//Function block to run a virtual drive with Nc
FUNCTION_BLOCK FB_Axis IMPLEMENTS I_axis
VAR
    _stAxis: REFERENCE TO ST_AxisStruct; // Local property pointer for axis structure
    astMcStatus: ARRAY[1..nMCSTATUS_ARRAY_SIZE] OF POINTER TO ST_McStatus; //Array of all MC status signals defined in FB_init

    fbPower: MC_Power;
    stMcStatusPower: ST_McStatus;

    fbStop: MC_Stop;
    stMcStatusStop: ST_McStatus;

    fbHalt: MC_Halt;
    stMcStatusHalt: ST_McStatus;

    fbReset: MC_Reset;
    stMcStatusReset: ST_McStatus;

    //SERCOS drive
    fbSoEReadDiagNumber : FB_SoEReadDiagNumber;
    fbSoEReset: FB_SoEReset;

    fbReadDriveInfo: FB_ReadDriveInfo;

    fbMoveAbsolute: MC_MoveAbsolute;
    fbMoveAbsolute2: MC_MoveAbsolute;
    stMcStatusMoveAbsolute: ST_McStatus;

    fbMoveRelative: MC_MoveRelative;
    stMcStatusMoveRelative: ST_McStatus;

    fbMoveVelocity: MC_MoveVelocity;
    stMcStatusMoveVelocity: ST_McStatus;

    fbMoveModulo: MC_MoveModulo;
    fbMoveModulo2: MC_MoveModulo;
    stMcStatusMoveModulo: ST_McStatus;

    fbBacklashCompensation: MC_BacklashCompensation;
    stMcStatusBacklash: ST_McStatus;

    fbHome: FB_Homing;
    stMcStatusHome: ST_McStatus;

    fbReadParameter: MC_ReadParameter;
    stMcStatusReadParameter: ST_McStatus;

    fbWriteParameter: MC_WriteParameter;
    stMcStatusWriteParameter: ST_McStatus;

    stMcStatusReadWriteCoE: ST_McStatus;
    fb_coe_writeEx: FB_EcCoESdoWriteEx; // Function Block for writing in CoE
    fb_coe_readEx: FB_EcCoESdoReadEx;  // Function Block for reading from CoE

    fbGearIn: MC_GearIn;
    stMcStatusGearIn: ST_McStatus;

    fbGearOut: MC_GearOut;
    stMcStatusGearOut: ST_McStatus;

    stMasterAxis: ST_GearAxis := (nIndex := 1, fRatio := 0);
    nSlaveAxesIndex: UINT;
    nAxisIndex: UINT;
    nMultiMastersAxesIndex: UINT;

    fbGearInMultiMaster: MC_GearInMultiMaster;
    stMcStatusGearInMultiMaster: ST_McStatus;

    //Custom made methods MC Status
    stMcStatusTempDisable: ST_McStatus;
    stMcStatusCommandHandler: ST_McStatus;
    stMcStatusAirpad: ST_McStatus;
    stMcStatusExternalBrake: ST_McStatus;

    //Variables for holding limits during homing
    bWaitForStopAfterLimitHit: BOOL := FALSE;
    fbRemovePowerTimer: TOF;

    //Dedicated NC parameter read FBs
    fbReadAxisVeloManSlow: MC_ReadParameter;
    fbReadAxisVeloManFast: MC_ReadParameter;
    fbReadHomingVelToCam: MC_ReadParameter;
    fbReadHomingVelFromCam: MC_ReadParameter;
    fbReadAxisVeloMax: MC_ReadParameter;
    fbReadAxisMaxAcc: MC_ReadParameter;
    fbReadAxisMaxDec: MC_ReadParameter;
    fbReadAxisAcc: MC_ReadParameter;
    fbReadAxisDec: MC_ReadParameter;
    fbReadEnMinSoftPosLimit: MC_ReadParameter;
    fbReadEnMaxSoftPosLimit: MC_ReadParameter;
    fbReadMinSoftPosLimit: MC_ReadParameter;
    fbReadMaxSoftPosLimit: MC_ReadParameter;
    fbReadEnPositionLagMonitoring: MC_ReadParameter;
    fbReadAxisMaxPosLagValue: MC_ReadParameter;
    fbReadEnTargetPositionMonitoring: MC_ReadParameter;
    fbReadTargetPositionWindow: MC_ReadParameter;
    fbReadBacklashConfigEnable: MC_ReadParameter;
    fbReadDriveAdress: MC_ReadDriveAddress;

    //Edge detection triggers for statuses
    fbDoneRTrig: R_TRIG;
    fbCommandAbortedRTrig: R_TRIG;
    fbInVelocityRTrig: R_TRIG;
    fbInVelocityFTrig: F_TRIG;
    fbExecuteRTrig: R_TRIG;
    fbStopFinishedRiseEdge: R_TRIG;
    fbHaltFinishedRiseEdge: R_TRIG;
    fbResetFinishedRiseEdge: R_TRIG;
    fbAbsMovDyn1RiseEdge: R_TRIG;
    fbAbsMovDyn2RiseEdge: R_TRIG;
    fbModMovDyn1RiseEdge: R_TRIG;
    fbModMovDyn2RiseEdge: R_TRIG;

    fbCommandHistory: FB_CommandHistory;

    bInternalExecute: BOOL := FALSE;
    bEnableCmdOld: BOOL := FALSE;
    bEnabledOld: BOOL := FALSE;
    bEnableAmpCmd: BOOL := FALSE;
END_VAR

VAR CONSTANT
    nRATIO_DENOMINATOR_DEFAULT: UINT := 1;
    nNO_GEARING: UINT := 0;
    nFIRST_ARRAY_INDEX_MOVE_COMMANDS: UINT := 5; //Used for the FOR loops for the Busy, Done, Command Aborted Status
    nLAST_ARRAY_INDEX_MOVE_COMMANDS: UINT := 15; //Used for the FOR loops for Done
    nMCSTATUS_ARRAY_SIZE: UINT := 19;
    nMULTI_MASTER_MAX_AXES: UINT := 4;
END_VAR

METHOD EndOfCycle : BOOL
IF _stAxis.stStatus.bDone
    OR _stAxis.stStatus.bError
    OR _stAxis.Axis.Status.Error
    OR _stAxis.Axis.Status.Disabled
    OR _stAxis.Axis.Status.Stopping
    OR _stAxis.stStatus.bCommandAborted
    OR NOT _stAxis.stStatus.bMoving THEN
    _stAxis.stStatus.eInternalMotionCommand := E_MotionFunctions.eWaitingForCommand;
END_IF

bInternalExecute := FALSE;
bEnabledOld := _stAxis.stStatus.bEnabled;
bEnableCmdOld := _stAxis.stControl.bEnable;

_stAxis.stControl.bExecute := FALSE;
END_METHOD

METHOD FB_init : BOOL
VAR_INPUT
    bInitRetains: BOOL; // if TRUE, the retain variables are initialized (warm start / cold start)
    bInCopyCode: BOOL; // if TRUE, the instance afterwards gets moved into the copy code (online change)
END_VAR
//Copy address locations for statuses to an array to allow for easier checking of statuses
astMcStatus[1] := ADR(stMcStatusPower);
astMcStatus[2] := ADR(stMcStatusStop);
astMcStatus[3] := ADR(stMcStatusHalt);
astMcStatus[4] := ADR(stMcStatusReset);
astMcStatus[5] := ADR(stMcStatusMoveAbsolute);
astMcStatus[6] := ADR(stMcStatusMoveRelative);
astMcStatus[7] := ADR(stMcStatusMoveVelocity);
astMcStatus[8] := ADR(stMcStatusMoveModulo);
astMcStatus[9] := ADR(stMcStatusHome);
astMcStatus[10] := ADR(stMcStatusGearInMultiMaster);
astMcStatus[11] := ADR(stMcStatusGearOut);
astMcStatus[12] := ADR(stMcStatusReadParameter);
astMcStatus[13] := ADR(stMcStatusWriteParameter);
astMcStatus[14] := ADR(stMcStatusReadWriteCoE);
astMcStatus[15] := ADR(stMcStatusBacklash);
astMcStatus[16] := ADR(stMcStatusTempDisable);
astMcStatus[17] := ADR(stMcStatusCommandHandler);
astMcStatus[18] := ADR(stMcStatusAirpad);
astMcStatus[19] := ADR(stMcStatusExternalBrake);
END_METHOD

// Controls pressure to airpad
METHOD mControl_Airpad : ST_McStatus
VAR_INPUT
    bMoveRequest: BOOL;
    bManualControl: BOOL;
    bManualPressureOn: BOOL;
END_VAR

VAR_OUTPUT
    bReady: BOOL;
END_VAR

VAR_INST
    eAirpad: E_Airpad := E_Airpad.eDepressurize;
    TON_PressurizeAirpad: TON;
    TON_Depressurize: TON;
    RTRIG_PressureRequest: R_TRIG;
    bNotPressurizedInTime: BOOL := FALSE;
    bPressureOnRequest: BOOL := FALSE;
    RTRIG_ManualControl: R_TRIG;

    nAirpadErrorId: UDINT := 0;
END_VAR
IF NOT _stAxis.stConfig.stAirpadBrake.bAirpadConnected THEN
    RETURN;
END_IF

RTRIG_ManualControl(CLK := _stAxis.stConfig.bAirpadManualControl);

IF RTRIG_ManualControl.Q THEN
    _stAxis.stControl.bAirpadManualPressureOn := bMoveRequest;
ELSIF NOT _stAxis.stConfig.bAirpadManualControl THEN
    _stAxis.stControl.bAirpadManualPressureOn := FALSE;
END_IF

bPressureOnRequest :=
    (bMoveRequest
        AND NOT bManualControl)
    OR (bManualControl
        AND bManualPressureOn);

RTRIG_PressureRequest(CLK := bPressureOnRequest);

TON_PressurizeAirpad(
    IN := bPressureOnRequest
        AND NOT _stAxis.stStatus.bError,
    PT := _stAxis.stConfig.stAirpadBrake.tAirpadOnDelayTime);

TON_Depressurize(
    IN := NOT bPressureOnRequest,
    PT := _stAxis.stConfig.stAirpadBrake.tAirpadOffDelayTime);

CASE eAirpad OF

    E_Airpad.eDepressurize:
        //No movement requested -> Airpad off
        _stAxis.stControl.bPressurizeAirpad := FALSE;
        IF bPressureOnRequest
            AND NOT _stAxis.stStatus.bError
            AND NOT _stAxis.stStatus.bAirpadPressureError THEN
            _stAxis.stStatus.bAirpadPressureError := FALSE;
            nAirpadErrorId := 0;
            eAirpad := E_Airpad.ePressurize;
        END_IF


    E_Airpad.ePressurize:
        //Movement requested -> Pressurize airpad
        _stAxis.stControl.bPressurizeAirpad := TRUE;

        IF _stAxis.stStatus.bError
            OR NOT bPressureOnRequest
            OR _stAxis.stStatus.bAirpadPressureError THEN
            eAirpad := E_Airpad.eDepressurize;
        ELSIF TON_PressurizeAirpad.Q THEN
            IF _stAxis.stConfig.stAirpadBrake.bAirpadFeedbackConnected
                AND NOT _stAxis.stInputs.bAirpadPressurized THEN
                _stAxis.stStatus.bAirpadPressureError := TRUE;
                nAirpadErrorId := E_CustomErrorIds.eAirPadPressureError;
                eAirpad := E_Airpad.eDepressurize;
            ELSE
                eAirpad := E_Airpad.eReadyToMove;
            END_IF
        END_IF


    E_Airpad.eReadyToMove:
        //Movement requested -> Airpad inflated
        _stAxis.stControl.bPressurizeAirpad := TRUE;

        IF _stAxis.stStatus.bError
            OR TON_Depressurize.Q
            OR _stAxis.stStatus.bAirpadPressureError THEN
            eAirpad := E_Airpad.eDepressurize;
        ELSIF (_stAxis.stConfig.stAirpadBrake.bAirpadFeedbackConnected
            AND NOT _stAxis.stInputs.bAirpadPressurized) THEN
            _stAxis.stStatus.bAirpadPressureError := TRUE;
            nAirpadErrorId := E_CustomErrorIds.eAirPadPressureError;
            eAirpad := E_Airpad.eDepressurize;
        END_IF

END_CASE

bReady := eAirpad = E_Airpad.eReadyToMove
    AND ((_stAxis.stConfig.stAirpadBrake.bAirpadFeedbackConnected
        AND _stAxis.stInputs.bAirpadPressurized)
    OR NOT _stAxis.stConfig.stAirpadBrake.bAirpadFeedbackConnected);

//ST_McStatus mapping
mControl_Airpad.Error := _stAxis.stStatus.bAirpadPressureError;
mControl_Airpad.ErrorID := nAirpadErrorId;

IF _stAxis.stStatus.bAirpadPressureError THEN
    _stAxis.stError.nAirpadErrorID := nAirpadErrorId;
END_IF
END_METHOD

METHOD mControl_BacklashCompensation : ST_McStatus
VAR_INPUT
END_VAR
(*Read Backlash documentation in the Confluence page or in Beckhoff before backlash setup:
https://confluence.ess.eu/display/MCAG/Backlash+compensation
Position compensation needs to be enabled in NC to use the backsash compensation*)

IF _stAxis.stConfig.stBacklashConfig.bEnabledInNC THEN

// Enabling the backlash functionality. It is disable if homing is performed.
    IF _stAxis.stStatus.bEnabled THEN
        IF fbHome.bBusy THEN
            fbBacklashCompensation.Enable := FALSE;
        ELSE
            fbBacklashCompensation.Enable := _stAxis.stConfig.stBacklashConfig.bEnableCompensation;
        END_IF
        fbBacklashCompensation.Backlash := _stAxis.stConfig.stBacklashConfig.fCorrectionSetting;
        fbBacklashCompensation.CompensationInPositiveDirection := _stAxis.stConfig.stBacklashConfig.bCompensationInPositiveDirection;
        fbBacklashCompensation.Ramp := ABS(_stAxis.stControl.fVelocity/3);
    ELSE
        fbBacklashCompensation.Enable := FALSE;
        fbBacklashCompensation.DisableMode := 1;
    END_IF

    fbBacklashCompensation(Axis := _stAxis.Axis);

END_IF

IF fbBacklashCompensation.Error THEN
    _stAxis.stError.nBacklashErrorID := fbBacklashCompensation.ErrorID;
END_IF
mControl_BacklashCompensation.Error := fbBacklashCompensation.Error;
mControl_BacklashCompensation.ErrorID := fbBacklashCompensation.ErrorID;
_stAxis.stStatus.bBacklashCompensating := fbBacklashCompensation.Limiting;
END_METHOD

// Handles delayed execution of motion commands due to e.g. auto-enable, airpad or external brake
METHOD mControl_CommandHandler : ST_McStatus

VAR_INPUT
    bAxisPermittedToMove: BOOL := FALSE;
    bPermitRequired: BOOL := FALSE;
END_VAR

VAR_OUTPUT
    bWaitingForMovePermit: BOOL;
    bMovePermit: BOOL;
    bReleaseMoveCmd: BOOL;
END_VAR

VAR
    bCommandAborted: BOOL;
END_VAR

VAR_INST
    eState: E_CommandHandlerState := E_CommandHandlerState.eIdle;
    eLatchedCommand: E_MotionFunctions;
    bInternalWaitingForMovePermit: BOOL := FALSE;
    bInternalMovePermit: BOOL := FALSE;
    bInternalReleasedMoveCmd: BOOL := FALSE;
    nWaitCounter: UINT := 0;
    RTRIG_Execute: R_TRIG;
    FTRIG_Moving: F_TRIG;
    TON_CommandHandlerTimeout: TON;
    RTRIG_ReleasedMoveCommand: R_TRIG;
    TON_LatchReleasedCommandStatus: TON;
    TON_DisableAxis: TON;
    RTRIG_DisableAxis: R_TRIG;
END_VAR
//State machine for command handling
RTRIG_Execute(CLK := _stAxis.stControl.bExecute);
RTRIG_ReleasedMoveCommand(CLK := bInternalReleasedMoveCmd);

CASE eState OF
    E_CommandHandlerState.eIdle:
        IF RTRIG_Execute.Q THEN
            CASE _stAxis.stControl.eCommand OF
                E_MotionFunctions.eMoveAbsolute,
                E_MotionFunctions.eMoveRelative,
                E_MotionFunctions.eMoveVelocity,
                E_MotionFunctions.eMoveModulo,
                E_MotionFunctions.eGearInMultiMaster,
                E_MotionFunctions.eGearOut,
                E_MotionFunctions.eHome :
                    eLatchedCommand := _stAxis.stControl.eCommand;
                    nWaitCounter := 0;
                    _stAxis.stStatus.bCommandHandlerTimeoutError := FALSE;

                    IF _stAxis.stConfig.bAutoEnable THEN
                        _stAxis.stControl.bEnable := TRUE;
                    END_IF

                    fbCommandHistory.mAdd(_stAxis.stControl);
                    eState := E_CommandHandlerState.eWaitPermits;
            END_CASE
        END_IF

    E_CommandHandlerState.eWaitPermits:
        IF (bPermitRequired AND bAxisPermittedToMove)
            OR NOT bPermitRequired
            OR (bPermitRequired AND NOT _stAxis.stConfig.bAutoEnable AND NOT _stAxis.stStatus.bEnabled) THEN

            eState := E_CommandHandlerState.eStabilizeNC;
        END_IF

    E_CommandHandlerState.eStabilizeNC:
        //Ensure permits are still valid during stabilization
        IF (bPermitRequired AND NOT bAxisPermittedToMove) THEN
             eState := E_CommandHandlerState.eWaitPermits;
             nWaitCounter := 0;
        ELSIF nWaitCounter >= _stAxis.stConfig.nCommandHandlerWaitCycles THEN
            eState := E_CommandHandlerState.eReleaseCommand;
        ELSE
            nWaitCounter := nWaitCounter + 1;
        END_IF

    E_CommandHandlerState.eReleaseCommand:
        _stAxis.stStatus.eInternalMotionCommand := eLatchedCommand;
        bInternalExecute := TRUE;
        bInternalMovePermit := TRUE;
        bInternalReleasedMoveCmd := TRUE;
        fbCommandHistory.mSetRelease();
        eState := E_CommandHandlerState.eWaitForMotionStart;

    E_CommandHandlerState.eWaitForMotionStart:
        IF _stAxis.stStatus.bMoving
            OR _stAxis.stStatus.bDone
            OR _stAxis.stStatus.bError THEN
            eState := E_CommandHandlerState.eIdle;
        END_IF

END_CASE

bInternalWaitingForMovePermit := (eState = E_CommandHandlerState.eWaitPermits OR eState = E_CommandHandlerState.eStabilizeNC);

TON_CommandHandlerTimeout(
    IN := bInternalWaitingForMovePermit,
    PT := _stAxis.stConfig.tCommandHandlerTimeout);

TON_LatchReleasedCommandStatus(IN := bInternalReleasedMoveCmd, PT := T#1S);

IF TON_CommandHandlerTimeout.Q THEN
    eState := E_CommandHandlerState.eIdle;
    bInternalWaitingForMovePermit := FALSE;
    bInternalMovePermit := FALSE;
    bInternalReleasedMoveCmd := FALSE;
    _stAxis.stStatus.bCommandHandlerTimeoutError := TRUE;
END_IF

IF _stAxis.stControl.bHalt
    OR _stAxis.stControl.bStop THEN
    bCommandAborted := bInternalWaitingForMovePermit;
    eState := E_CommandHandlerState.eIdle;
    bInternalWaitingForMovePermit := FALSE;
    bInternalMovePermit := FALSE;
    bInternalReleasedMoveCmd := FALSE;
END_IF

FTRIG_Moving(CLK :=
    (_stAxis.stStatus.bMoving AND NOT _stAxis.Axis.Status.HomingBusy)
    OR _stAxis.Axis.Status.HomingBusy);

IF FTRIG_Moving.Q
    OR _stAxis.stStatus.bError THEN
    eState := E_CommandHandlerState.eIdle;
    bInternalWaitingForMovePermit := FALSE;
    bInternalMovePermit := FALSE;
    bInternalReleasedMoveCmd := FALSE;
END_IF

TON_DisableAxis(
    IN := _stAxis.stConfig.bAutoDisable
        AND _stAxis.stStatus.bEnabled
        AND NOT bInternalWaitingForMovePermit
        AND NOT bInternalMovePermit
        AND NOT bInternalReleasedMoveCmd,
    PT := _stAxis.stConfig.tAutoDisableHysteresis);
RTRIG_DisableAxis(CLK := TON_DisableAxis.Q);
IF RTRIG_DisableAxis.Q
    AND _stAxis.stConfig.bAutoDisable THEN
    _stAxis.stControl.bEnable := FALSE;
END_IF

IF RTRIG_ReleasedMoveCommand.Q THEN
    bInternalReleasedMoveCmd := TRUE;
END_IF

IF TON_LatchReleasedCommandStatus.Q THEN
    bInternalReleasedMoveCmd := FALSE;
END_IF

bWaitingForMovePermit := bInternalWaitingForMovePermit;
bMovePermit := bInternalMovePermit;
bReleaseMoveCmd := bInternalReleasedMoveCmd;

mControl_CommandHandler.CommandAborted := bCommandAborted;
mControl_CommandHandler.Done := bInternalExecute;
mControl_CommandHandler.Busy := (eState <> E_CommandHandlerState.eIdle);
mControl_CommandHandler.Error := _stAxis.stStatus.bCommandHandlerTimeoutError;

IF _stAxis.stStatus.bCommandHandlerTimeoutError THEN
    mControl_CommandHandler.ErrorID := TO_UDINT(E_CustomErrorIds.eCommandHandlerTimeoutError);
    _stAxis.stError.nCommandHandlerErrorID := mControl_CommandHandler.ErrorID;
END_IF
END_METHOD

// Controls external brake
METHOD mControl_ExternalBrake: BOOL

VAR_OUTPUT
    bReady: BOOL;
END_VAR

VAR_INST
    eExternalBrake: E_ExternalBrake := E_ExternalBrake.eBrakeEngaged;
    bEnableAmp: BOOL := FALSE;
    TON_DelayBrakeRelease: TON;
    TON_DelayAmplifierDisable: TON;
    bStartDelayBrakeOpening: BOOL := FALSE;
    bStartDelayAmplifierDisable: BOOL := FALSE;
    bStartBrakeOpeningTimeout: BOOL := FALSE;
    TON_BrakeOpeningTimeoutWhenFeedback: TON;
END_VAR
IF _stAxis.stControl.bEnable AND NOT bEnableCmdOld
    AND NOT _stAxis.stStatus.bExternalBrakeFailure THEN
    eExternalBrake := E_ExternalBrake.eDelayBrakeRelease;
    bStartDelayBrakeOpening := FALSE;
    _stAxis.stStatus.bExternalBrakeTimeoutError  := FALSE;
END_IF

IF (NOT _stAxis.stControl.bEnable OR _stAxis.stStatus.bError)
    AND bEnableCmdOld THEN
    eExternalBrake := E_ExternalBrake.eCloseBrakeDelayAmplifier;
    bStartDelayAmplifierDisable := FALSE;
END_IF

TON_DelayBrakeRelease(
    IN := bStartDelayBrakeOpening,
    PT := _stAxis.stConfig.stAirpadBrake.tBrakeOpenDelayTime
);

TON_DelayAmplifierDisable(
    IN := bStartDelayAmplifierDisable,
    PT := _stAxis.stConfig.stAirpadBrake.tBrakeCloseAheadTime
);

TON_BrakeOpeningTimeoutWhenFeedback(
    IN := bStartBrakeOpeningTimeout,
    PT := _stAxis.stConfig.stAirpadBrake.tBrakeOpeningTimeoutWhenFeedback
);

IF TON_BrakeOpeningTimeoutWhenFeedback.Q THEN
    _stAxis.stStatus.bExternalBrakeTimeoutError := TRUE;
END_IF

CASE eExternalBrake OF

    E_ExternalBrake.eBrakeEngaged:
        _stAxis.stControl.bReleaseBrake := FALSE;
        bStartDelayBrakeOpening := FALSE;
        bStartDelayAmplifierDisable := FALSE;
        bStartBrakeOpeningTimeout := FALSE;
        bEnableAmp := FALSE;


    E_ExternalBrake.eDelayBrakeRelease:
        // Postpone opening of brake
        bEnableAmp := TRUE;
        bStartDelayAmplifierDisable := FALSE;

        IF TON_DelayBrakeRelease.Q THEN
            IF NOT _stAxis.stStatus.bEnabled
                OR _stAxis.stStatus.bError
                OR TON_BrakeOpeningTimeoutWhenFeedback.Q THEN
                _stAxis.stControl.bEnable := FALSE;
                _stAxis.stControl.bReleaseBrake := FALSE;
                bEnableAmp := FALSE;
                eExternalBrake := E_ExternalBrake.eBrakeEngaged;
            ELSE
                _stAxis.stControl.bReleaseBrake := TRUE;
                bStartBrakeOpeningTimeout := TRUE;
            END_IF

            IF _stAxis.stControl.bReleaseBrake
                AND ((_stAxis.stConfig.stAirpadBrake.bExternalBrakeFeedbackConnected
                    AND _stAxis.stInputs.bBrakeReleased)
                OR NOT _stAxis.stConfig.stAirpadBrake.bExternalBrakeFeedbackConnected) THEN
                eExternalBrake := E_ExternalBrake.eBrakeReleased;
                bStartBrakeOpeningTimeout := FALSE;
            END_IF
        END_IF

        // If enabled lost while opening, go directly to closed
        IF bEnabledOld
            AND (NOT _stAxis.stStatus.bEnabled OR _stAxis.stStatus.bError) THEN
            eExternalBrake := E_ExternalBrake.eBrakeEngaged;
            bEnableAmp := FALSE;
            _stAxis.stControl.bReleaseBrake := FALSE;
        END_IF

        // Start counting when enabled
        IF _stAxis.stStatus.bEnabled
            AND eExternalBrake <> E_ExternalBrake.eBrakeReleased THEN
            bStartDelayBrakeOpening := TRUE;
        END_IF


    E_ExternalBrake.eBrakeReleased:
        bStartDelayBrakeOpening := FALSE;
        bStartDelayAmplifierDisable := FALSE;
        // If enabled lost, or if brake feedback fails: go directly to closed
        IF (NOT _stAxis.stStatus.bEnabled OR _stAxis.stStatus.bError)
            AND _stAxis.stControl.bEnable THEN
            _stAxis.stControl.bReleaseBrake := FALSE;
            _stAxis.stControl.bEnable := FALSE;
            bEnableAmp := FALSE;
            eExternalBrake := E_ExternalBrake.eBrakeEngaged;
        ELSIF _stAxis.stConfig.stAirpadBrake.bExternalBrakeFeedbackConnected
            AND _stAxis.stControl.bReleaseBrake
            AND NOT _stAxis.stInputs.bBrakeReleased THEN
            _stAxis.stControl.bReleaseBrake := FALSE;
            _stAxis.stControl.bEnable := FALSE;
            bEnableAmp := FALSE;
            eExternalBrake := E_ExternalBrake.eBrakeEngaged;
            _stAxis.stStatus.bExternalBrakeFailure := TRUE;
        ELSE
            _stAxis.stControl.bReleaseBrake := TRUE;
            bEnableAmp := TRUE;
        END_IF


    // The check for bError in first rows of this function changes state to eCloseBrakeDelayAmplifier.
    // If bError TRUE we directly disable amplifier. Good?
    // Might be good to also perform a check of the bSTOComing signal:
    // * bStOComing -> wait for axis stopped -> eBrakeCloseDelayAmplifier
    // If STO comes before eBrakeClosed -> the detection of bErrorStop should take us into eBrakeClosed.
    E_ExternalBrake.eCloseBrakeDelayAmplifier:
        // Postpone disabling of amplifier
        _stAxis.stControl.bReleaseBrake := FALSE;
        bStartDelayBrakeOpening := FALSE;
        bStartDelayAmplifierDisable := TRUE;
        bEnableAmp := TRUE;
        IF TON_DelayAmplifierDisable.Q
            OR NOT _stAxis.stStatus.bEnabled
            OR _stAxis.stStatus.bError THEN
            eExternalBrake := E_ExternalBrake.eBrakeEngaged;
            bEnableAmp := FALSE;
        END_IF

END_CASE

bReady :=
    eExternalBrake = E_ExternalBrake.eBrakeReleased
    AND ((_stAxis.stConfig.stAirpadBrake.bExternalBrakeFeedbackConnected
        AND _stAxis.stInputs.bBrakeReleased)
    OR NOT _stAxis.stConfig.stAirpadBrake.bExternalBrakeFeedbackConnected);
mControl_ExternalBrake := bEnableAmp;
END_METHOD

METHOD mControl_GearInMultiMaster : ST_McStatus
fbGearInMultiMaster.Options.AdvancedSlaveDynamics := TRUE;
fbGearInMultiMaster.Options.SyncMode := E_GearInMultiMasterSyncMode.POSSYNC2;
IF _stAxis.stControl.eCommand = E_MotionFunctions.eGearInMultiMaster THEN
    fbGearInMultiMaster.Enable := _stAxis.stControl.bExecute;
END_IF

IF _stAxis.stControl.eCommand = E_MotionFunctions.eGearInMultiMaster AND _stAxis.stControl.bExecute AND NOT _stAxis.Axis.Status.Coupled THEN
    //Latch master references
    FOR nMultiMastersAxesIndex := 1 TO nMULTI_MASTER_MAX_AXES DO
        IF _stAxis.stConfig.astMultiMasterAxis[nMultiMastersAxesIndex].nIndex > 0 AND _stAxis.stConfig.astMultiMasterAxis[nMultiMastersAxesIndex].nIndex <= GVL_APP.nAXIS_NUM THEN
            _stAxis.stConfig.astMultiMasterAxisLatched[nMultiMastersAxesIndex].nIndex := _stAxis.stConfig.astMultiMasterAxis[nMultiMastersAxesIndex].nIndex;
        END_IF
    END_FOR
    //Latch gear ratios
    FOR nMultiMastersAxesIndex := 1 TO nMULTI_MASTER_MAX_AXES DO
        _stAxis.stConfig.astMultiMasterAxisLatched[nMultiMastersAxesIndex].fRatio := _stAxis.stConfig.astMultiMasterAxis[nMultiMastersAxesIndex].fRatio;
    END_FOR
    //Transfer gear ratios to FB
    fbGearInMultiMaster.GearRatio1 := _stAxis.stConfig.astMultiMasterAxisLatched[1].fRatio;
    fbGearInMultiMaster.GearRatio2 := _stAxis.stConfig.astMultiMasterAxisLatched[2].fRatio;
    fbGearInMultiMaster.GearRatio3 := _stAxis.stConfig.astMultiMasterAxisLatched[3].fRatio;
    fbGearInMultiMaster.GearRatio4 := _stAxis.stConfig.astMultiMasterAxisLatched[4].fRatio;
    fbGearInMultiMaster.Enable := TRUE;
END_IF

fbGearInMultiMaster(Slave := _stAxis.Axis,
    Master1 := GVL.astAxes[_stAxis.stConfig.astMultiMasterAxisLatched[1].nIndex].Axis,
    Master2 := GVL.astAxes[_stAxis.stConfig.astMultiMasterAxisLatched[2].nIndex].Axis,
    Master3 := GVL.astAxes[_stAxis.stConfig.astMultiMasterAxisLatched[3].nIndex].Axis,
    Master4 := GVL.astAxes[_stAxis.stConfig.astMultiMasterAxisLatched[4].nIndex].Axis);
fbGearInMultiMaster.Enable:= FALSE;

IF fbGearInMultiMaster.InGear THEN
    mStatus_MultiGearing();
END_IF

IF fbGearInMultiMaster.Error THEN
    fbGearInMultiMaster.Enable := FALSE;
END_IF

mControl_GearInMultiMaster.Active := fbGearInMultiMaster.Active;
mControl_GearInMultiMaster.Done := fbGearInMultiMaster.InGear;
mControl_GearInMultiMaster.Busy := fbGearInMultiMaster.Busy;
mControl_GearInMultiMaster.Error := fbGearInMultiMaster.Error;
mControl_GearInMultiMaster.ErrorID := fbGearInMultiMaster.ErrorID;
mControl_GearInMultiMaster.CommandAborted := fbGearInMultiMaster.CommandAborted;

IF fbGearInMultiMaster.Error THEN
    _stAxis.stError.nGearInMultiMasterErrorID := fbGearInMultiMaster.ErrorID; //Set the error
END_IF

fbCommandHistory.mSetResultOfCommand(
    eCommand := E_MotionFunctions.eGearInMultiMaster,
    stStatus := mControl_GearInMultiMaster);
END_METHOD

METHOD mControl_GearOut : ST_McStatus
IF _stAxis.stControl.eCommand = E_MotionFunctions.eGearOut THEN
    fbGearOut.Execute := _stAxis.stControl.bExecute;
END_IF

fbGearOut(Slave := _stAxis.Axis);
fbGearOut.Execute := FALSE;

//Clear ratios from single and multi master gearing
IF fbGearOut.Done THEN
    //Clear slave ratio from master axis slave array
    mStatus_MultiGearing();
    FOR nSlaveAxesIndex := 1 TO GVL_APP.nAXIS_NUM DO
        GVL.astAxes[nSlaveAxesIndex].stConfig.afMultiSlaveAxisRatio[GVL.iAxis] := nNO_GEARING;
    END_FOR
END_IF

mControl_GearOut.Done := fbGearOut.Done;
mControl_GearOut.Busy := fbGearOut.Busy;
mControl_GearOut.Error := fbGearOut.Error;
mControl_GearOut.ErrorID := fbGearOut.ErrorID;

IF fbGearOut.Error THEN
    _stAxis.stError.nGearOutErrorID := fbGearOut.ErrorID; //Set the error
END_IF

fbCommandHistory.mSetResultOfCommand(
    eCommand := E_MotionFunctions.eGearOut,
    stStatus := mControl_GearOut);
END_METHOD

METHOD mControl_Home : ST_McStatus
IF _stAxis.stConfig.eHomeSeq = E_HomingRoutines.eNoHoming THEN
    _stAxis.stStatus.bHomed := TRUE;
END_IF

IF _stAxis.stStatus.eInternalMotionCommand = E_MotionFunctions.eHome THEN
    fbHome.bExecute := bInternalExecute;
END_IF


fbHome.eHomingRoutine := _stAxis.stConfig.eHomeSeq;
fbHome.fHomePosition := _stAxis.stConfig.fHomePosition;
fbHome.fHomeFinishDistance := _stAxis.stConfig.fHomeFinishDistance;
fbHome(
    Axis := _stAxis.Axis,
    bLimitBwd := _stAxis.stInputs.bLimitBwd,
    bLimitFwd := _stAxis.stInputs.bLimitFwd,
    bHomeSensor := _stAxis.stInputs.bHomeSensor,
    stConfig := _stAxis.stConfig.stHomingConfig);
fbHome.bExecute := FALSE;

mControl_Home.Busy := fbHome.bBusy;
mControl_Home.CommandAborted := fbHome.bCommandAborted;
mControl_Home.Done := fbHome.bDone;
mControl_Home.Error := fbHome.bError;
mControl_Home.ErrorID := fbHome.nErrorId;

IF fbHome.bError THEN
    _stAxis.stError.nHomeErrorID := fbHome.nErrorID; //Set the error
END_IF

fbCommandHistory.mSetResultOfCommand(
    eCommand := E_MotionFunctions.eHome,
    stStatus := mControl_Home);
END_METHOD

METHOD mControl_LimitHitTimer : BOOL
//Timer for keeping power on after limit switch hit, needed for homing routines - if power is lost routines are aborted
fbRemovePowerTimer(IN := _stAxis.stInputs.bLimitFwd AND _stAxis.stInputs.bLimitBwd, PT := T#100MS);

IF stMcStatusHome.Busy AND (fbRemovePowerTimer.Q OR _stAxis.Axis.NcToPlc.AxisState = 5) THEN //5=PHASE_ACCNEG
    bWaitForStopAfterLimitHit := TRUE;
ELSE
    bWaitForStopAfterLimitHit := FALSE;
END_IF
END_METHOD

METHOD mControl_LimitLinking : BOOL
(*Linking Fwd/BwdEnabled. Fwd and Bwd can e.g. be enabled by its respective limit
switches or by both of them (this is normally only during first commissioning*)

_stAxis.stStatus.bFwEnabled :=
    (_stAxis.stInputs.bLimitFwd
    AND (_stAxis.stInputs.bLimitBwd OR NOT _stAxis.stConfig.bEnableStopWithAnyLimitSwitch)
    OR bWaitForStopAfterLimitHit)
    AND NOT _stAxis.stStatus.bInterlockedFwd
    AND _stAxis.stStatus.bAxisReadyToMove;
_stAxis.stStatus.bBwEnabled :=
    (_stAxis.stInputs.bLimitBwd
    AND (_stAxis.stInputs.bLimitFwd OR NOT _stAxis.stConfig.bEnableStopWithAnyLimitSwitch)
    OR bWaitForStopAfterLimitHit)
    AND NOT _stAxis.stStatus.bInterlockedBwd
    AND _stAxis.stStatus.bAxisReadyToMove;

_stAxis.stStatus.bInterlockedFwd := _stAxis.stControl.bInterlockFwd;
_stAxis.stStatus.bInterlockedBwd := _stAxis.stControl.bInterlockBwd;

//Multimaster limit linking
FOR nAxisIndex := 1 TO GVL_APP.nAXIS_NUM DO
    IF _stAxis.stConfig.afMultiSlaveAxisRatio[nAxisIndex] <> 0 THEN
        _stAxis.stStatus.bFwEnabled :=
            _stAxis.stStatus.bFwEnabled
            AND SEL(_stAxis.stConfig.afMultiSlaveAxisRatio[nAxisIndex] > 0,
                GVL.astAxes[nAxisIndex].stStatus.bBwEnabled,
                GVL.astAxes[nAxisIndex].stStatus.bFwEnabled);
        _stAxis.stStatus.bBwEnabled :=
            _stAxis.stStatus.bBwEnabled
            AND SEL(_stAxis.stConfig.afMultiSlaveAxisRatio[nAxisIndex] > 0,
                GVL.astAxes[nAxisIndex].stStatus.bFwEnabled,
                GVL.astAxes[nAxisIndex].stStatus.bBwEnabled);
    END_IF
END_FOR
END_METHOD

METHOD mControl_Power : ST_McStatus
stMcStatusTempDisable := mControl_TemperatureDisable(_stAxis.stConfig.bEnableTemperatureDisable);
IF  _stAxis.stStatus.bHighTempAxisDisabled THEN
    _stAxis.stControl.bEnable := FALSE;
END_IF

IF _stAxis.stConfig.stAirpadBrake.bExternalBrakeConnected THEN
    bEnableAmpCmd :=
        mControl_ExternalBrake(bReady => _stAxis.stStatus.bExternalBrakeReady);
ELSE
    bEnableAmpCmd := _stAxis.stControl.bEnable;
END_IF

fbPower.Enable := bEnableAmpCmd;

fbPower.Enable_Negative := _stAxis.stStatus.bBwEnabled OR (bEnableAmpCmd AND fbHome.bEnableNegative);

fbPower.Enable_Positive := _stAxis.stStatus.bFwEnabled OR (bEnableAmpCmd AND fbHome.bEnablePositive);

fbPower.Override := _stAxis.stConfig.fOverride;

fbPower(Axis := _stAxis.Axis);

mControl_Power.Error := fbPower.Error;

IF fbPower.Error THEN
    _stAxis.stError.nPowerErrorID := fbPower.ErrorID; //Set the error
END_IF
END_METHOD

METHOD mControl_Reset : ST_McStatus
VAR
    i: UINT;
END_VAR
VAR_INST
    bSoEReset: BOOL := FALSE;
END_VAR
(*The function block MC_Reset is used to reset the NC axis. In many cases this also leads
to a reset of a connected drive device. Depending on the bus system or drive types,
in some cases a separate reset may be required for the drive device.*)

IF _stAxis.stControl.bReset
    AND _stAxis.stConfig.stDriveInfo.DeviceType = E_DeviceType.DEVICETYPE_SOE_DEFAULT
    AND NOT fbReset.Busy THEN
    bSoEReset := TRUE;
    fbSoEReset.Execute := bSoEReset;
END_IF

fbSoEReset(Axis := _stAxis.Axis);

IF bSoEReset
    AND NOT fbSoEReset.Busy THEN
    fbSoEReset.Execute := FALSE;
    bSoEReset := FALSE;
END_IF

IF NOT fbSoEReset.Busy THEN
    fbReset.Execute := _stAxis.stControl.bReset;
END_IF

fbReset(Axis := _stAxis.Axis);

IF fbReset.Done
    AND NOT bSoEReset
    AND NOT fbSoEReset.Busy THEN
    _stAxis.stStatus.bError := FALSE;
    _stAxis.stStatus.bCommandHandlerTimeoutError := FALSE;
    _stAxis.stStatus.bAirpadPressureError := FALSE;
    _stAxis.stStatus.bExternalBrakeTimeoutError := FALSE;
    _stAxis.stStatus.bExternalBrakeFailure := FALSE;
    FOR i := 1 TO nMCSTATUS_ARRAY_SIZE DO
        astMcStatus[i]^.Error := FALSE;
        astMcStatus[i]^.ErrorID := 0;
    END_FOR
    //Reset ST_Status error ID
    _stAxis.stStatus.nErrorID := 0;
    //Reset St_AxisError error IDs (MEMSET ensures future additions are automatically handled)
    MEMSET(ADR(_stAxis.stError), 0, SIZEOF(_stAxis.stError));

END_IF

mControl_Reset.Busy := fbReset.Busy OR fbSoEReset.Busy;
mControl_Reset.Done := fbReset.Done AND NOT fbSoEReset.Busy;
mControl_Reset.Error := fbReset.Error OR fbSoEReset.Error;
mControl_Reset.ErrorID := fbReset.ErrorID;

IF fbReset.Error THEN
    _stAxis.stError.nResetErrorID := fbReset.ErrorID; //Set the error
END_IF

fbResetFinishedRiseEdge(CLK:=fbReset.Done OR fbReset.Error);
IF fbResetFinishedRiseEdge.Q OR fbReset.Done THEN
    _stAxis.stControl.bReset := FALSE;
END_IF
END_METHOD

METHOD mControl_TemperatureDisable: ST_McStatus
VAR_INPUT
    bEnableTemperatureDisable: BOOL;
END_VAR

VAR
    nAxisId: DINT;
END_VAR

VAR_INST
    rTrigErrorMessage: R_TRIG;
    fbErrorMessageTON: TON;
    fTemperatureScaledValue: REAL;
    fTemperatureValue: REAL;
    bResetErrorMessage: BOOL;
    bTempSensorError: BOOL := FALSE;
    nErrorID: UDINT := 0;
END_VAR

VAR CONSTANT
    fDISCONNECTED_VALUE: REAL := 850.0;
    fWRONG_CONNECTION_VALUE: REAL := -200.0;
END_VAR
nAxisId := UDINT_TO_DINT(_stAxis.Axis.NcToPlc.AxisId);
rTrigErrorMessage(CLK := bResetErrorMessage);
fTemperatureScaledValue := INT_TO_REAL(_stAxis.stInputs.nTempPT100)/_stAxis.stConfig.fTempScalingFactor;
fTemperatureValue := SEL(_stAxis.stControl.bHWMaskActive,
    fTemperatureScaledValue,
    _stAxis.stControl.fMaskedTemperature);
fbErrorMessageTON(IN := bResetErrorMessage, PT:=T#30M);

_stAxis.stStatus.fActTemperature := fTemperatureValue;

IF NOT bEnableTemperatureDisable THEN
    RETURN;
END_IF

bTempSensorError := fTemperatureValue >= fDISCONNECTED_VALUE
    OR fTemperatureValue <= fWRONG_CONNECTION_VALUE;

//Check for disconnection or wrongly connected errors
IF bTempSensorError THEN
    nErrorID := E_CustomErrorIds.eTemperatureSensorError;
    bResetErrorMessage := TRUE;
    _stAxis.stStatus.bHighTempAxisDisabled := TRUE;

    IF rTrigErrorMessage.Q THEN
        IF fTemperatureValue = fDISCONNECTED_VALUE THEN
            ADSLOGDINT(msgCtrlMask := ADSLOG_MSGTYPE_ERROR,
                msgFmtStr := 'ERROR: Temperature sensor of Axis %d is disconnected.',
                dintArg := nAxisId);
        ELSIF fTemperatureValue = fWRONG_CONNECTION_VALUE THEN
            ADSLOGDINT(msgCtrlMask := ADSLOG_MSGTYPE_ERROR,
                msgFmtStr := 'ERROR: Temperature sensor of Axis %d is wrongly connected, check pin connections.',
                dintArg := nAxisId);
        END_IF
    END_IF

    //Reset bError to display Error message every 30 minutes if error is still there
    IF fbErrorMessageTON.Q THEN
        bResetErrorMessage := FALSE;
    END_IF
ELSE
    nErrorID := E_CustomErrorIds.eNoCustomError;
    IF fTemperatureValue < _stAxis.stConfig.fMaxTemperature AND NOT _stAxis.stStatus.bHighTempAxisDisabled THEN
        bResetErrorMessage := FALSE;
        _stAxis.stStatus.bHighTempAxisDisabled := FALSE;
    ELSIF fTemperatureValue < _stAxis.stConfig.fMaxTemperature AND _stAxis.stStatus.bHighTempAxisDisabled THEN
        IF fTemperatureValue <= (_stAxis.stConfig.fMaxTemperature - 5.0) THEN
            _stAxis.stStatus.bHighTempAxisDisabled := FALSE;
            bResetErrorMessage := FALSE;
        ELSE
            bResetErrorMessage := TRUE;
        END_IF
    ELSIF fTemperatureValue >= _stAxis.stConfig.fMaxTemperature THEN
        bResetErrorMessage := TRUE;
        _stAxis.stStatus.bHighTempAxisDisabled := TRUE;
        IF rTrigErrorMessage.Q THEN
            ADSLOGDINT(msgCtrlMask := ADSLOG_MSGTYPE_ERROR,
                msgFmtStr := 'ERROR: Axis temperature too hot. Axis %d was disabled.',
                dintArg := nAxisId);
        END_IF

        IF fbErrorMessageTON.Q THEN
            bResetErrorMessage := FALSE;
        END_IF
    END_IF
END_IF

_stAxis.stStatus.bTempSensorError := bTempSensorError;

mControl_TemperatureDisable.Active := bEnableTemperatureDisable;
mControl_TemperatureDisable.Error := bTempSensorError;
mControl_TemperatureDisable.ErrorID := nErrorID;

IF bTempSensorError THEN
    _stAxis.stError.nTempDisableErrorID := nErrorID;
END_IF
END_METHOD

METHOD mMove_Halt : ST_McStatus
fbHalt.Deceleration := _stAxis.stControl.fDeceleration;
fbHalt.Execute := _stAxis.stControl.bHalt;

fbHalt(Axis := _stAxis.Axis);

mMove_Halt.Busy := fbHalt.Busy;
mMove_Halt.Done := fbHalt.Done;
mMove_Halt.Error := fbHalt.Error;
mMove_Halt.ErrorID := fbHalt.ErrorID;
mMove_Halt.Active := fbHalt.Active;
mMove_Halt.CommandAborted := fbHalt.CommandAborted;

fbCommandHistory.mSetHalted(bExecute := fbHalt.Execute);

IF fbHalt.Error THEN
    _stAxis.stError.nHaltErrorID := fbHalt.ErrorID; //Set the error
END_IF

//Execution of fbHalt ended
fbHaltFinishedRiseEdge(CLK:=fbHalt.Done OR fbHalt.Error OR fbHalt.CommandAborted);
IF fbHaltFinishedRiseEdge.Q OR fbHalt.Done OR fbHalt.CommandAborted THEN
    _stAxis.stControl.bHalt := FALSE;
END_IF
END_METHOD

METHOD mMove_MoveAbsolute : ST_McStatus
IF _stAxis.stStatus.eInternalMotionCommand = E_MotionFunctions.eMoveAbsolute THEN
    fbMoveAbsolute.Execute := bInternalExecute;
    IF fbMoveAbsolute.Execute AND fbMoveAbsolute.Busy THEN
        fbMoveAbsolute2.Execute := TRUE;
    END_IF
END_IF

// Parameters
fbMoveAbsolute.Position := _stAxis.stControl.fPosition;
fbMoveAbsolute.Velocity := ABS(_stAxis.stControl.fVelocity);
fbMoveAbsolute.Acceleration := _stAxis.stControl.fAcceleration;
fbMoveAbsolute.Deceleration := _stAxis.stControl.fDeceleration;

fbMoveAbsolute2.Position := _stAxis.stControl.fPosition;
fbMoveAbsolute2.Velocity := ABS(_stAxis.stControl.fVelocity);
fbMoveAbsolute2.Acceleration := _stAxis.stControl.fAcceleration;
fbMoveAbsolute2.Deceleration := _stAxis.stControl.fDeceleration;


// Call both move absolute FB
fbMoveAbsolute(Axis := _stAxis.Axis);
fbMoveAbsolute2(Axis := _stAxis.Axis);

//Reset Execute bits
fbMoveAbsolute.Execute := FALSE;
fbMoveAbsolute2.Execute := FALSE;

// STATUS bits
mMove_MoveAbsolute.Active := fbMoveAbsolute.Active OR fbMoveAbsolute2.Active;
mMove_MoveAbsolute.Done := fbMoveAbsolute.Done OR fbMoveAbsolute2.Done;
mMove_MoveAbsolute.Busy := fbMoveAbsolute.Busy OR fbMoveAbsolute2.Busy;
mMove_MoveAbsolute.Error := fbMoveAbsolute.Error OR fbMoveAbsolute2.Error;

// Capture the CommandAborted for first scan if the other absolute move overtakes the current
fbAbsMovDyn1RiseEdge(CLK:= fbMoveAbsolute.Busy AND fbMoveAbsolute2.CommandAborted, Q=>);
fbAbsMovDyn2RiseEdge(CLK:= fbMoveAbsolute2.Busy AND fbMoveAbsolute.CommandAborted, Q=>);
mMove_MoveAbsolute.CommandAborted := (fbMoveAbsolute.CommandAborted AND NOT fbAbsMovDyn2RiseEdge.Q)
                                    OR (fbMoveAbsolute2.CommandAborted AND NOT fbAbsMovDyn1RiseEdge.Q);

// Error IDs
IF fbMoveAbsolute.Error THEN
    _stAxis.stError.nMoveAbsoluteErrorID := fbMoveAbsolute.ErrorID; //Set the error
    mMove_MoveAbsolute.ErrorID := fbMoveAbsolute.ErrorID;
END_IF
IF fbMoveAbsolute2.Error THEN
    _stAxis.stError.nMoveAbsoluteErrorID := fbMoveAbsolute2.ErrorID; //Set the error
    mMove_MoveAbsolute.ErrorID := fbMoveAbsolute2.ErrorID;
END_IF

fbCommandHistory.mSetResultOfCommand(
    eCommand := E_MotionFunctions.eMoveAbsolute,
    stStatus := mMove_MoveAbsolute);
END_METHOD

METHOD mMove_MoveModulo : ST_McStatus
IF _stAxis.stStatus.eInternalMotionCommand = E_MotionFunctions.eMoveModulo THEN
    fbMoveModulo.Execute := bInternalExecute;
    IF fbMoveModulo.Execute AND fbMoveModulo.Busy THEN
        fbMoveModulo2.Execute := TRUE;
    END_IF
END_IF

// Parameters
fbMoveModulo.Position := _stAxis.stControl.fPosition;
fbMoveModulo.Velocity := ABS(_stAxis.stControl.fVelocity);
fbMoveModulo.Acceleration := _stAxis.stControl.fAcceleration;
fbMoveModulo.Deceleration := _stAxis.stControl.fDeceleration;

fbMoveModulo2.Position := _stAxis.stControl.fPosition;
fbMoveModulo2.Velocity := ABS(_stAxis.stControl.fVelocity);
fbMoveModulo2.Acceleration := _stAxis.stControl.fAcceleration;
fbMoveModulo2.Deceleration := _stAxis.stControl.fDeceleration;

// Call both move absolute FB
fbMoveModulo(Axis := _stAxis.Axis);
fbMoveModulo.Execute := FALSE;
fbMoveModulo2(Axis := _stAxis.Axis);
fbMoveModulo2.Execute := FALSE;

// Status bits
mMove_MoveModulo.Active := fbMoveModulo.Active OR fbMoveModulo2.Active;
mMove_MoveModulo.Done := fbMoveModulo.Done OR fbMoveModulo2.Done;
mMove_MoveModulo.Busy := fbMoveModulo.Busy OR fbMoveModulo2.Busy;
mMove_MoveModulo.Error := fbMoveModulo.Error OR fbMoveModulo2.Error;

// Capture the CommandAborted for first scan if the other absolute move overtakes the current
fbModMovDyn1RiseEdge(CLK:= fbMoveModulo.Busy AND fbMoveModulo2.CommandAborted, Q=>);
fbModMovDyn2RiseEdge(CLK:= fbMoveModulo2.Busy AND fbMoveModulo.CommandAborted, Q=>);
mMove_MoveModulo.CommandAborted := (fbMoveModulo.CommandAborted AND NOT fbModMovDyn2RiseEdge.Q)
                                    OR (fbMoveModulo2.CommandAborted AND NOT fbModMovDyn1RiseEdge.Q);

// Error IDs
IF fbMoveModulo.Error THEN
    _stAxis.stError.nMoveModuloErrorID := fbMoveModulo.ErrorID; //Set the error
    mMove_MoveModulo.ErrorID := fbMoveModulo.ErrorID;
END_IF

IF fbMoveModulo2.Error THEN
    _stAxis.stError.nMoveModuloErrorID := fbMoveModulo2.ErrorID; //Set the error
    mMove_MoveModulo.ErrorID := fbMoveModulo2.ErrorID;
END_IF

fbCommandHistory.mSetResultOfCommand(
    eCommand := E_MotionFunctions.eMoveModulo,
    stStatus := mMove_MoveModulo);
END_METHOD

METHOD mMove_MoveRelative : ST_McStatus
IF _stAxis.stStatus.eInternalMotionCommand = E_MotionFunctions.eMoveRelative THEN
    fbMoveRelative.Execute := bInternalExecute;
END_IF

fbMoveRelative.Distance := _stAxis.stControl.fPosition;
fbMoveRelative.Velocity := ABS(_stAxis.stControl.fVelocity);
fbMoveRelative.Acceleration := _stAxis.stControl.fAcceleration;
fbMoveRelative.Deceleration := _stAxis.stControl.fDeceleration;

fbMoveRelative(Axis := _stAxis.Axis);
fbMoveRelative.Execute := FALSE;

mMove_MoveRelative.Active := fbMoveRelative.Active;
mMove_MoveRelative.Done := fbMoveRelative.Done;
mMove_MoveRelative.Busy := fbMoveRelative.Busy;
mMove_MoveRelative.Error := fbMoveRelative.Error;
mMove_MoveRelative.ErrorID := fbMoveRelative.ErrorID;
mMove_MoveRelative.CommandAborted := fbMoveRelative.CommandAborted;

IF fbMoveRelative.Error THEN
    _stAxis.stError.nMoveRelativeErrorID := fbMoveRelative.ErrorID; //Set the error
END_IF

fbCommandHistory.mSetResultOfCommand(
    eCommand := E_MotionFunctions.eMoveRelative,
    stStatus := mMove_MoveRelative);
END_METHOD

METHOD mMove_MoveVelocity : ST_McStatus
IF _stAxis.stStatus.eInternalMotionCommand = E_MotionFunctions.eMoveVelocity THEN
    fbMoveVelocity.Execute := bInternalExecute;
END_IF

fbMoveVelocity.Direction := SEL(_stAxis.stControl.fVelocity < 0, MC_Positive_Direction, MC_Negative_Direction);
fbMoveVelocity.Velocity := ABS(_stAxis.stControl.fVelocity);
fbMoveVelocity.Acceleration := _stAxis.stControl.fAcceleration;
fbMoveVelocity.Deceleration := _stAxis.stControl.fDeceleration;

fbMoveVelocity(Axis := _stAxis.Axis);
fbMoveVelocity.Execute:= FALSE;

mMove_MoveVelocity.Active := fbMoveVelocity.Active;
mMove_MoveVelocity.InVelocity := fbMoveVelocity.InVelocity;
mMove_MoveVelocity.Busy := fbMoveVelocity.Busy;
mMove_MoveVelocity.Error := fbMoveVelocity.Error;
mMove_MoveVelocity.ErrorID := fbMoveVelocity.ErrorID;
mMove_MoveVelocity.CommandAborted := fbMoveVelocity.CommandAborted;

IF fbMoveVelocity.Error THEN
    _stAxis.stError.nMoveVelocityErrorID := fbMoveVelocity.ErrorID; //Set the error
END_IF

fbCommandHistory.mSetResultOfCommand(
    eCommand := E_MotionFunctions.eMoveVelocity,
    stStatus := mMove_MoveVelocity);
END_METHOD

METHOD mMove_Stop : ST_McStatus
fbStop.Deceleration := _stAxis.stControl.fDeceleration;
fbStop.Execute := _stAxis.stControl.bStop;

fbStop(Axis := _stAxis.Axis);

mMove_Stop.Busy := fbStop.Busy;
mMove_Stop.Done := fbStop.Done;
mMove_Stop.Error := fbStop.Error;
mMove_Stop.ErrorID := fbStop.ErrorID;
mMove_Stop.Active := fbStop.Active;
mMove_Stop.CommandAborted := fbStop.CommandAborted;

fbCommandHistory.mSetStopped(bExecute := fbStop.Execute);

IF fbStop.Error THEN
    _stAxis.stError.nStopErrorID := fbStop.ErrorID; //Set the error
END_IF

//Execution of fbStop ended
fbStopFinishedRiseEdge(CLK:=fbStop.Done OR fbStop.Error OR fbStop.CommandAborted);
IF fbStopFinishedRiseEdge.Q THEN
    _stAxis.stControl.bStop := FALSE;
END_IF
END_METHOD

METHOD mParameters_Init : BOOL
VAR_INST
    FTRIG_DriveBusy: F_TRIG;
    bInitializeDriveInfo: BOOL := TRUE;
    bInitializeParameters: BOOL := TRUE;
    nInitializeDriveCounter: UINT := 0;
END_VAR
IF _stAxis.stConfig.bReadMcParametersValid
    AND bInitializeParameters THEN
    _stAxis.stControl.fAcceleration := _stAxis.stConfig.fDefaultAcc;
    _stAxis.stControl.fDeceleration := _stAxis.stConfig.fDefaultDec;
    _stAxis.stControl.fVelocity := _stAxis.stConfig.fVelocityDefaultFast;
    _stAxis.stControl.fJogVelocity := _stAxis.stConfig.fVelocityDefaultSlow;

    bInitializeParameters := FALSE;
END_IF

IF bInitializeDriveInfo
    AND NOT bInitializeParameters THEN
    FTRIG_DriveBusy(CLK := fbReadDriveInfo.Busy);

    IF FTRIG_DriveBusy.Q THEN
        bInitializeDriveInfo := FALSE;
    END_IF

    fbReadDriveInfo(
        Axis := _stAxis.Axis,
        Execute := bInitializeDriveInfo,
        DriveInfo => _stAxis.stConfig.stDriveInfo);

    // Retry if error
    IF NOT bInitializeDriveInfo
        AND fbReadDriveInfo.Error
        AND nInitializeDriveCounter < 3 THEN
        bInitializeDriveInfo := TRUE;
        nInitializeDriveCounter := nInitializeDriveCounter + 1;
    END_IF
END_IF

_stAxis.stStatus.bAxisInitialized :=
    NOT bInitializeParameters AND NOT bInitializeDriveInfo;
END_METHOD

METHOD mParameters_ReadNc : BOOL
(*This act reads the MC parameters using an MC_ReadParameter FB FOR each variable
Intended TO be executed once every PLC cycle
Another FB is used TO trasnfer default axis parameters TO the stAxisStruct so
bReadValid is used TO halt that trasnfer UNTIL the parameters have been
read successfully. It may take a couple OF cycles once the PLC starts up.*)

//Slow jogging Velocity
fbReadAxisVeloManSlow(Axis := _stAxis.Axis,
                        Enable := TRUE,
                        ReadMode := READMODE_CYCLIC,
                        ParameterNumber := E_AxisParameters.AxisManualVelocitySlow,
                        Value => _stAxis.stConfig.fVelocityDefaultSlow);
//Fast jogging velocity
fbReadAxisVeloManFast(Axis := _stAxis.Axis,
                        Enable := TRUE,
                        ReadMode := READMODE_CYCLIC,
                        ParameterNumber := E_AxisParameters.AxisManualVelocityFast,
                        Value => _stAxis.stConfig.fVelocityDefaultFast);
//Homing velocity to Cam
fbReadHomingVelToCam(Axis := _stAxis.Axis,
                        Enable := TRUE,
                        ReadMode := READMODE_CYCLIC,
                        ParameterNumber := E_AxisParameters.AxisVelocityToCam,
                        Value => _stAxis.stConfig.fHomingVelToCam);
//Homing velocity from Cam
fbReadHomingVelFromCam(Axis := _stAxis.Axis,
                        Enable := TRUE,
                        ReadMode := READMODE_CYCLIC,
                        ParameterNumber := E_AxisParameters.AxisVelocityFromCam,
                        Value => _stAxis.stConfig.fHomingVelFromCam);
//Max velocity
fbReadAxisVeloMax(Axis := _stAxis.Axis,
                        Enable := TRUE,
                        ReadMode := READMODE_CYCLIC,
                        ParameterNumber := E_AxisParameters.AxisMaxVelocity,
                        Value => _stAxis.stConfig.fVeloMax);
//Max acceleration
fbReadAxisMaxAcc(Axis := _stAxis.Axis,
                        Enable := TRUE,
                        ReadMode := READMODE_CYCLIC,
                        ParameterNumber := E_AxisParameters.AxisMaximumAcceleration,
                        Value => _stAxis.stConfig.fMaxAcc);
//Max deceleration
fbReadAxisMaxDec(Axis := _stAxis.Axis,
                        Enable := TRUE,
                        ReadMode := READMODE_CYCLIC,
                        ParameterNumber := E_AxisParameters.AxisMaximumDeceleration,
                        Value => _stAxis.stConfig.fMaxDec);
//Default acceleration
fbReadAxisAcc(Axis := _stAxis.Axis,
                        Enable := TRUE,
                        ReadMode := READMODE_CYCLIC,
                        ParameterNumber := E_AxisParameters.AxisDefaultAcceleration,
                        Value => _stAxis.stConfig.fDefaultAcc);
//Default deceleration
fbReadAxisDec(Axis := _stAxis.Axis,
                        Enable := TRUE,
                        ReadMode := READMODE_CYCLIC,
                        ParameterNumber := E_AxisParameters.AxisDefaultDeceleration,
                        Value => _stAxis.stConfig.fDefaultDec);

//Soft limits enabled
fbReadEnMinSoftPosLimit(Axis := _stAxis.Axis,
                        Enable := TRUE,
                        ReadMode := READMODE_CYCLIC,
                        ParameterNumber := E_AxisParameters.EnableLimitBackward);
_stAxis.stConfig.bEnMinSoftPosLimit := LREAL_TO_BOOL(fbReadEnMinSoftPosLimit.Value);

fbReadEnMaxSoftPosLimit(Axis := _stAxis.Axis,
                        Enable := TRUE,
                        ReadMode := READMODE_CYCLIC,
                        ParameterNumber := E_AxisParameters.EnableLimitForward);
_stAxis.stConfig.bEnMaxSoftPosLimit := LREAL_TO_BOOL(fbReadEnMaxSoftPosLimit.Value);

//Soft limit values
fbReadMinSoftPosLimit(Axis := _stAxis.Axis,
                        Enable := TRUE,
                        ReadMode := READMODE_CYCLIC,
                        ParameterNumber := E_AxisParameters.SWLimitBackward,
                        Value => _stAxis.stConfig.fMinSoftPosLimit);
fbReadMaxSoftPosLimit(Axis := _stAxis.Axis,
                        Enable := TRUE,
                        ReadMode := READMODE_CYCLIC,
                        ParameterNumber := E_AxisParameters.SWLimitForward,
                        Value => _stAxis.stConfig.fMaxSoftPosLimit);

//Position Lag Monitoring
fbReadEnPositionLagMonitoring(Axis := _stAxis.Axis,
                        Enable := TRUE,
                        ReadMode := READMODE_CYCLIC,
                        ParameterNumber := E_AxisParameters.EnablePositionLagMonitoring);
_stAxis.stConfig.bEnPositionLagMonitoring := LREAL_TO_BOOL(fbReadEnPositionLagMonitoring.Value);

fbReadAxisMaxPosLagValue(Axis := _stAxis.Axis,
                        Enable := TRUE,
                        ReadMode := READMODE_CYCLIC,
                        ParameterNumber := E_AxisParameters.MaxPositionLag,
                        Value => _stAxis.stConfig.fMaxPosLagValue);

// Target Position Monitoring
fbReadEnTargetPositionMonitoring(Axis := _stAxis.Axis,
                        Enable := TRUE,
                        ReadMode := READMODE_CYCLIC,
                        ParameterNumber := E_AxisParameters.SWLimitBackward);
_stAxis.stConfig.bEnTargetPositionMonitoring := LREAL_TO_BOOL(fbReadEnTargetPositionMonitoring.Value);

fbReadTargetPositionWindow(Axis := _stAxis.Axis,
                        Enable := TRUE,
                        ReadMode := READMODE_CYCLIC,
                        ParameterNumber := E_AxisParameters.AxisTargetPositionWindow,
                        Value => _stAxis.stConfig.fTargetPositionWindow);

// Position Compensation
fbReadBacklashConfigEnable(Axis := _stAxis.Axis,
                        Enable := TRUE,
                        ReadMode := READMODE_CYCLIC,
                        ParameterNumber := E_AxisParameters.AxisEnablePosCorrection);
_stAxis.stConfig.stBacklashConfig.bEnabledInNC := LREAL_TO_BOOL(fbReadBacklashConfigEnable.Value);


//All variables are valid
_stAxis.stConfig.bReadMcParametersValid := FALSE;
_stAxis.stConfig.bReadMcParametersValid := fbReadAxisVeloManSlow.Valid AND
    fbReadAxisVeloManFast.Valid AND
    fbReadHomingVelToCam.Valid AND
    fbReadHomingVelFromCam.Valid AND
    fbReadAxisVeloMax.Valid AND
    fbReadAxisAcc.Valid AND
    fbReadAxisDec.Valid AND
    fbReadEnMinSoftPosLimit.Valid AND
    fbReadEnMaxSoftPosLimit.Valid AND
    fbReadMinSoftPosLimit.Valid AND
    fbReadMaxSoftPosLimit.Valid AND
    fbReadEnPositionLagMonitoring.Valid AND
    fbReadAxisMaxPosLagValue.Valid AND
    fbReadEnTargetPositionMonitoring.Valid AND
    fbReadTargetPositionWindow.Valid;

//One of the variables has a read error
_stAxis.stConfig.bReadMcParametersError := fbReadAxisVeloManSlow.Error OR
    fbReadAxisVeloManFast.Error OR
    fbReadHomingVelToCam.Error OR
    fbReadHomingVelFromCam.Error OR
    fbReadAxisVeloMax.Error OR
    fbReadAxisAcc.Error OR
    fbReadAxisDec.Error OR
    fbReadEnMinSoftPosLimit.Error OR
    fbReadEnMaxSoftPosLimit.Error OR
    fbReadMinSoftPosLimit.Error OR
    fbReadMaxSoftPosLimit.Error OR
    fbReadEnPositionLagMonitoring.Error OR
    fbReadAxisMaxPosLagValue.Error OR
    fbReadEnTargetPositionMonitoring.Error OR
    fbReadTargetPositionWindow.Error;
END_METHOD

METHOD mParameters_ReadParameter : ST_McStatus
IF _stAxis.stControl.eCommand = E_MotionFunctions.eReadParameter THEN
    fbReadParameter.Enable := _stAxis.stControl.bExecute;
END_IF

fbReadParameter.ReadMode := E_READMODE.READMODE_ONCE;
{warning disable C0327} // Disable compiler warning 'Implicit conversion from enumeration to another'
fbReadParameter.ParameterNumber := _stAxis.stConfig.eAxisParameters;
{warning restore C0327}

fbReadParameter(Axis := _stAxis.Axis);
fbReadParameter.Enable := FALSE;

_stAxis.stconfig.fReadAxisParameter := fbReadParameter.Value;
mParameters_ReadParameter.Busy := fbReadParameter.Busy;
mParameters_ReadParameter.Done := fbReadParameter.Valid;
mParameters_ReadParameter.Error := fbReadParameter.Error;
mParameters_ReadParameter.ErrorID := fbReadParameter.ErrorID;

IF fbReadParameter.Error THEN
    _stAxis.stError.nReadParameterErrorId := fbReadParameter.ErrorID;
END_IF
END_METHOD

METHOD PUBLIC mParameters_ReadWriteCoE : ST_McStatus
CASE _stAxis.stConfig.stCoEParameters.nState OF

// ============== INIT , READ ADRESS=================
E_CoEParamState.eInit:
    fbReadDriveAdress(Axis := _stAxis.Axis, Execute := _stAxis.stStatus.bAxisInitialized);
    IF fbReadDriveAdress.Done THEN
        _stAxis.stConfig.stCoEParameters.sEthCATNetId := fbReadDriveAdress.DriveAddress.NetID;
        _stAxis.stConfig.stCoEParameters.nSlaveAdressDrive := fbReadDriveAdress.DriveAddress.SlaveAddress;
        fbReadDriveAdress.Execute := FALSE;
        _stAxis.stConfig.stCoEParameters.nState := E_CoEParamState.eIdle; //skip read name  for now...
    ELSIF fbReadDriveAdress.Error THEN
        _stAxis.stConfig.stCoEParameters.nState := E_CoEParamState.eError;     // Error case
        mParameters_ReadWriteCoE.ErrorID := fbReadDriveAdress.ErrorID;
        fbReadDriveAdress.Execute := FALSE;
    END_IF


    E_CoEParamState.eReadName: //Read device name
        fb_coe_readex(
           sNetId:= _stAxis.stConfig.stCoEParameters.sEthCATNetId,
           nSlaveAddr:= (_stAxis.stConfig.stCoEParameters.nSlaveAdressDrive),
           nSubIndex:= 0, //Device name without sub-index number
           nIndex:= INT_TO_WORD(16#1008),
           pDstBuf:= ADR(_stAxis.stConfig.stCoEParameters.sDeviceName),
           cbBufLen:= 80,
           bExecute:= TRUE,
           tTimeout:= T#1S,
           bCompleteAccess := FALSE
           );
        IF fb_coe_readex.bError THEN
          _stAxis.stConfig.stCoEParameters.nState := E_CoEParamState.eError;
        ELSIF NOT fb_coe_readex.bBusy THEN
          _stAxis.stConfig.stCoEParameters.nState := E_CoEParamState.eIdle;
          fb_coe_readex(bExecute := FALSE);
        END_IF

    E_CoEParamState.eIdle:
       IF _stAxis.stControl.eCommand = E_MotionFunctions.eWriteCoEParameters AND _stAxis.stControl.bExecute THEN
          //Prepare CoE-Access: Write value of CoE object/ sub index:
          fb_coe_writeex(bExecute := FALSE);
          _stAxis.stConfig.stCoEParameters.nState := E_CoEParamState.eWriteStart; //Next state for writing
       END_IF
       IF _stAxis.stControl.eCommand = E_MotionFunctions.eReadCoEParameters AND _stAxis.stControl.bExecute THEN
          //Prepare CoE-Access: Read value of CoE object/ sub index:
          fb_coe_readex(bExecute := FALSE);
          _stAxis.stConfig.stCoEParameters.nState := E_CoEParamState.eReadDriveParam; //Next state for reading
       END_IF
       _stAxis.stConfig.stCoEParameters.bDone := FALSE;

    E_CoEParamState.eWriteStart:
       //Write entry
       fb_coe_writeEx(
       sNetId:= _stAxis.stConfig.stCoEParameters.sEthCATNetId,
       nSlaveAddr:= (_stAxis.stConfig.stCoEParameters.nSlaveAdressDrive),
       nSubIndex:= INT_TO_BYTE(_stAxis.stConfig.stCoEParameters.eCoEParameters),
       nIndex:= _stAxis.stConfig.stCoEParameters.nIndexDrive,
       pSrcBuf:= ADR(_stAxis.stConfig.stCoEParameters.aParWrite),
       cbBufLen:= 2,
       bExecute:= TRUE,
       tTimeout:= T#1S,
       bCompleteAccess := FALSE
       );
       _stAxis.stConfig.stCoEParameters.nState := E_CoEParamState.eWriteWaitingForDone;

    E_CoEParamState.eWriteWaitingForDone:
       //Execute CoE write until done
       fb_coe_writeEx();
       IF fb_coe_writeEx.bError THEN
          _stAxis.stConfig.stCoEParameters.nState := E_CoEParamState.eError;
       ELSE
           IF NOT fb_coe_writeEx.bBusy THEN
                fb_coe_writeEx(bExecute := FALSE);
                _stAxis.stConfig.stCoEParameters.bDone := TRUE;
                _stAxis.stConfig.stCoEParameters.nState := E_CoEParamState.eIdle;
           END_IF
       END_IF

    E_CoEParamState.eReadDriveParam:
        IF _stAxis.stConfig.stCoEParameters.nSlaveAdressDrive <>0 THEN
            IF _stAxis.stConfig.stCoEParameters.nIndexDrive <>0 THEN
                IF NOT fb_coe_readEx.bExecute THEN
                    // Read entry
                    fb_coe_readEx(
                       sNetId:= _stAxis.stConfig.stCoEParameters.sEthCATNetId,
                       nSlaveAddr:= (_stAxis.stConfig.stCoEParameters.nSlaveAdressDrive),
                       nSubIndex:= INT_TO_BYTE(_stAxis.stConfig.stCoEParameters.eCoEParameters),
                       nIndex:= (_stAxis.stConfig.stCoEParameters.nIndexDrive),
                       pDstBuf:= ADR(_stAxis.stConfig.stCoEParameters.aParRead),
                       cbBufLen:= 2,
                       bExecute:= TRUE,
                       tTimeout:= T#1S,
                       bCompleteAccess := FALSE
                       );
                END_IF
                    fb_coe_readEx();//Execute CoE read until done
                    IF fb_coe_readEx.bError THEN
                        _stAxis.stConfig.stCoEParameters.nState := E_CoEParamState.eError;
                    ELSE
                    IF NOT fb_coe_readEx.bBusy THEN
                        fb_coe_readEx(bExecute := FALSE);
                        _stAxis.stConfig.stCoEParameters.bDone := TRUE;
                        _stAxis.stConfig.stCoEParameters.nState := E_CoEParamState.eIdle;
                    END_IF
                END_IF
            END_IF
        ELSE
            _stAxis.stConfig.stCoEParameters.nState := E_CoEParamState.eError;     // Error case
        END_IF

// ============== COE ERROR =================
E_CoEParamState.eError:
    // Error handling..
    IF _stAxis.stControl.bReset THEN
        _stAxis.stConfig.stCoEParameters.nState := E_CoEParamState.eIdle;
    END_IF
   ;
END_CASE

mParameters_ReadWriteCoE.Busy := fb_coe_writeex.bBusy OR fb_coe_readex.bBusy;
mParameters_ReadWriteCoE.Done := _stAxis.stConfig.stCoEParameters.bDone;
mParameters_ReadWriteCoE.Error := fb_coe_readex.bError OR fb_coe_writeex.bError OR _stAxis.stConfig.stCoEParameters.nState = E_CoEParamState.eError;
IF fb_coe_readex.bError THEN
    mParameters_ReadWriteCoE.ErrorID := fb_coe_readex.nErrId;
ELSIF fb_coe_writeex.bError THEN
    mParameters_ReadWriteCoE.ErrorID := fb_coe_writeex.nErrId;
ELSIF _stAxis.stConfig.stCoEParameters.nState = E_CoEParamState.eError THEN
    mParameters_ReadWriteCoE.ErrorID := 7;
END_IF
END_METHOD

METHOD mParameters_WriteParameter : ST_McStatus
IF _stAxis.stControl.eCommand = E_MotionFunctions.eWriteParameter THEN
    fbWriteParameter.Execute := _stAxis.stControl.bExecute;
END_IF

{warning disable C0327} // Disable compiler warning 'Implicit conversion from enumeration to another'
fbWriteParameter.ParameterNumber := _stAxis.stConfig.eAxisParameters;
{warning restore C0327}
fbWriteParameter.Value := _stAxis.stConfig.fWriteAxisParameter;

fbWriteParameter(Axis := _stAxis.Axis);
fbWriteParameter.Execute := FALSE;

mParameters_WriteParameter.Busy := fbWriteParameter.Busy;
mParameters_WriteParameter.Done := fbWriteParameter.Done;
mParameters_WriteParameter.Error := fbWriteParameter.Error;
mParameters_WriteParameter.ErrorID := fbWriteParameter.ErrorID;

IF fbWriteParameter.Error THEN
    _stAxis.stError.nWriteParameterErrorId := fbWriteParameter.ErrorID;
END_IF
END_METHOD

METHOD mStatus_AxisStatus : BOOL

VAR_INST
    rtrigBwdLimit: R_TRIG;
    ftrigBwdLimit: F_TRIG;
    rtrigFwdLimit: R_TRIG;
    ftrigFwdLimit: F_TRIG;

    rtrigHomeSensor: R_TRIG;
    ftrigHomeSensor: F_TRIG;
END_VAR
_stAxis.Axis.ReadStatus();
IF _stAxis.Axis.Status.OpMode.Modulo THEN
    _stAxis.stStatus.fActPosition := _stAxis.Axis.NcToPlc.ModuloActPos;
ELSE
    _stAxis.stStatus.fActPosition := _stAxis.Axis.NcToPlc.ActPos;
END_IF

_stAxis.stStatus.bGeared := _stAxis.Axis.Status.Coupled;
_stAxis.stStatus.bHomed := _stAxis.Axis.Status.Homed;
_stAxis.stStatus.bMoving := _stAxis.Axis.Status.Moving;
_stAxis.stStatus.fActVelocity := _stAxis.Axis.NcToPlc.ActVelo;
_stAxis.stStatus.bMovingForward := _stAxis.Axis.Status.PositiveDirection;
_stAxis.stStatus.bMovingBackward := _stAxis.Axis.Status.NegativeDirection;
_stAxis.stStatus.bInTargetPosition := _stAxis.Axis.Status.InTargetPosition;
_stAxis.stStatus.bSoEDriveDeviceError := _stAxis.Axis.Status.DriveDeviceError;
_stAxis.stStatus.bEnabled := NOT(_stAxis.Axis.Status.Disabled);

{info 'NOTE: The fuses controlling the outputs are currently not monitored, constituting a risk for an airpad/brake without feedback.'}
_stAxis.stStatus.bAxisReadyToMove := _stAxis.stStatus.bEnabled
    AND (NOT _stAxis.stConfig.stAirpadBrake.bAirpadConnected
        OR (_stAxis.stControl.bPressurizeAirpad AND _stAxis.stStatus.bAirpadReady))
    AND (NOT _stAxis.stConfig.stAirpadBrake.bExternalBrakeConnected
        OR (_stAxis.stControl.bReleaseBrake AND _stAxis.stStatus.bExternalBrakeReady));

_stAxis.stError.nNCErrorID := _stAxis.Axis.Status.ErrorID;

rtrigBwdLimit(CLK := _stAxis.stInputs.bLimitBwd);
ftrigBwdLimit(CLK := _stAxis.stInputs.bLimitBwd);
rtrigFwdLimit(CLK := _stAxis.stInputs.bLimitFwd);
ftrigFwdLimit(CLK := _stAxis.stInputs.bLimitFwd);

rtrigHomeSensor(CLK := _stAxis.stInputs.bHomeSensor);
ftrigHomeSensor(CLK := _stAxis.stInputs.bHomeSensor);

IF NOT _stAxis.stStatus.bAxisInitialized THEN
    RETURN;
END_IF

//The switch is expected to be true when not engaged.
IF ftrigBwdLimit.Q THEN
    _stAxis.stStatus.stSwitchInfo.fLimitBwdTrigPos := _stAxis.stStatus.fActPosition;
    _stAxis.stStatus.stSwitchInfo.nLimitBwdTrigEncoderRaw := _stAxis.stStatus.nEncoderRawCounter;
    _stAxis.stStatus.stSwitchInfo.fLimitBwdTrigExternalPos := _stAxis.stInputs.fExternalPos;
END_IF

IF rtrigBwdLimit.Q THEN
    _stAxis.stStatus.stSwitchInfo.fLimitBwdUntrigPos := _stAxis.stStatus.fActPosition;
    _stAxis.stStatus.stSwitchInfo.nLimitBwdUntrigEncoderRaw := _stAxis.stStatus.nEncoderRawCounter;
    _stAxis.stStatus.stSwitchInfo.fLimitBwdUntrigExternalPos := _stAxis.stInputs.fExternalPos;
END_IF

IF ftrigFwdLimit.Q THEN
    _stAxis.stStatus.stSwitchInfo.fLimitFwdTrigPos := _stAxis.stStatus.fActPosition;
    _stAxis.stStatus.stSwitchInfo.nLimitFwdTrigEncoderRaw := _stAxis.stStatus.nEncoderRawCounter;
    _stAxis.stStatus.stSwitchInfo.fLimitFwdTrigExternalPos := _stAxis.stInputs.fExternalPos;
END_IF

IF rtrigFwdLimit.Q THEN
    _stAxis.stStatus.stSwitchInfo.fLimitFwdUntrigPos := _stAxis.stStatus.fActPosition;
    _stAxis.stStatus.stSwitchInfo.nLimitFwdUntrigEncoderRaw := _stAxis.stStatus.nEncoderRawCounter;
    _stAxis.stStatus.stSwitchInfo.fLimitFwdUntrigExternalPos := _stAxis.stInputs.fExternalPos;
END_IF

IF rtrigHomeSensor.Q THEN
    _stAxis.stStatus.stSwitchInfo.fHomeSensorTrigPos := _stAxis.stStatus.fActPosition;
    _stAxis.stStatus.stSwitchInfo.nHomeSensorTrigEncoderRaw := _stAxis.stStatus.nEncoderRawCounter;
    _stAxis.stStatus.stSwitchInfo.fHomeSensorTrigExternalPos := _stAxis.stInputs.fExternalPos;
END_IF

IF ftrigHomeSensor.Q THEN
    _stAxis.stStatus.stSwitchInfo.fHomeSensorUntrigPos := _stAxis.stStatus.fActPosition;
    _stAxis.stStatus.stSwitchInfo.nHomeSensorUntrigEncoderRaw := _stAxis.stStatus.nEncoderRawCounter;
    _stAxis.stStatus.stSwitchInfo.fHomeSensorUntrigExternalPos := _stAxis.stInputs.fExternalPos;
END_IF
END_METHOD

METHOD mStatus_Busy : BOOL
VAR
    i: UINT;
    tmpBusy: BOOL;
END_VAR
FOR i := nFIRST_ARRAY_INDEX_MOVE_COMMANDS TO nMCSTATUS_ARRAY_SIZE DO
    tmpBusy := astMcStatus[i]^.Busy OR tmpBusy;
END_FOR
mStatus_Busy := tmpBusy;
END_METHOD

METHOD mStatus_CommandAborted : BOOL
VAR
    i: UINT;
    tmpCmdAborted: BOOL;
END_VAR
FOR i := nFIRST_ARRAY_INDEX_MOVE_COMMANDS TO nMCSTATUS_ARRAY_SIZE DO
    tmpCmdAborted := astMcStatus[i]^.CommandAborted OR tmpCmdAborted;
END_FOR

fbCommandAbortedRTrig(CLK := tmpCmdAborted);
IF fbCommandAbortedRTrig.Q THEN
    _stAxis.stStatus.bCommandAborted := TRUE;
END_IF
END_METHOD

METHOD mStatus_Done : BOOL
VAR
    i: UINT;
    tmpDone: BOOL;
END_VAR
FOR i := nFIRST_ARRAY_INDEX_MOVE_COMMANDS TO nLAST_ARRAY_INDEX_MOVE_COMMANDS DO
    tmpDone := astMcStatus[i]^.Done OR tmpDone;
END_FOR
//fbDoneRTrig(CLK:= mStatus_Done());
fbDoneRTrig(CLK := tmpDone);
IF fbDoneRTrig.Q THEN
    _stAxis.stStatus.bDone := TRUE;
END_IF
END_METHOD

METHOD mStatus_Error : BOOL
VAR
    i: UINT;
END_VAR
IF _stAxis.stConfig.stDriveInfo.DeviceType = E_DeviceType.DEVICETYPE_SOE_DEFAULT THEN
    // Read SERCOS drive error information,
    fbSoEReadDiagNumber(
        Axis := stAxis.Axis,
        Execute :=TRUE,
        Timeout := DEFAULT_ADS_TIMEOUT,
        SercosErrId => stAxis.stStatus.nSoEErrorID,
        DiagNumber => stAxis.stStatus.nSoEDiagID);

    IF NOT fbSoEReadDiagNumber.Busy THEN
        fbSoEReadDiagNumber(Axis := stAxis.Axis, Execute := FALSE);
    END_IF
ELSE
    stAxis.stStatus.nSoEErrorID := 0;
    stAxis.stStatus.nSoEDiagID := 0;
END_IF

//Evaluate overall axis error, default to the NC's ErrorStop status
_stAxis.stStatus.bError := _stAxis.Axis.Status.ErrorStop;

//Override with TRUE if any custom method has an error
FOR i := (nLAST_ARRAY_INDEX_MOVE_COMMANDS + 1) TO nMCSTATUS_ARRAY_SIZE DO
    IF astMcStatus[i]^.Error THEN
        _stAxis.stStatus.bError := TRUE;
    END_IF
END_FOR

//Allow nErrorID to be set only if 0, to create a snapshot of the root cause.
IF _stAxis.stStatus.nErrorID = 0 THEN
    //Set the NC Error ID as a baseline fallback
    IF _stAxis.Axis.Status.ErrorStop THEN
        _stAxis.stStatus.nErrorID := _stAxis.Axis.Status.ErrorID;
    ELSIF _stAxis.Axis.Status.Error THEN
        _stAxis.stStatus.nErrorID := _stAxis.stError.nNCErrorID;
    END_IF

    //Overwrite with FB/Custom Errors if present.
    //Because this executes after the NC check, the FB error gets priority.
    FOR i := 1 TO nMCSTATUS_ARRAY_SIZE DO
        IF astMcStatus[i]^.Error AND astMcStatus[i]^.ErrorID <> 0 THEN
            _stAxis.stStatus.nErrorID := astMcStatus[i]^.ErrorID;
            EXIT;
        END_IF
    END_FOR
END_IF
END_METHOD

METHOD mStatus_InVelocity : BOOL
VAR
    i: UINT;
    tmpInVelocity: BOOL;
END_VAR
FOR i := 1 TO nMCSTATUS_ARRAY_SIZE DO
    tmpInVelocity := astMcStatus[i]^.InVelocity OR tmpInVelocity;
END_FOR
//fbInVelocityRTrig(CLK:= mStatus_InVelocity());
fbInVelocityRTrig(CLK := tmpInVelocity);
IF fbInVelocityRTrig.Q THEN
    _stAxis.stStatus.bInVelocity := TRUE;
END_IF

fbInVelocityFTrig(CLK := _stAxis.Axis.Status.ContinuousMotion);
IF fbInVelocityFTrig.Q THEN
    _stAxis.stStatus.bInVelocity := FALSE;
END_IF
END_METHOD

METHOD mStatus_MultiGearing : BOOL
IF _stAxis.Axis.Status.Coupled AND _stAxis.Axis.PlcToNc.GearRatio1 <> 0 AND _stAxis.stConfig.astMultiMasterAxisLatched[1].nIndex <> 0 THEN
    GVL.astAxes[_stAxis.stConfig.astMultiMasterAxisLatched[1].nIndex].stConfig.afMultiSlaveAxisRatio[GVL.iAxis] := _stAxis.Axis.PlcToNc.GearRatio1;
    _stAxis.stStatus.bCoupledGear1 := TRUE;
ELSE
    _stAxis.stStatus.bCoupledGear1 := FALSE;
END_IF

IF _stAxis.Axis.Status.Coupled AND _stAxis.Axis.PlcToNc.GearRatio2 <> 0 AND _stAxis.stConfig.astMultiMasterAxisLatched[2].nIndex <> 0 THEN
    GVL.astAxes[_stAxis.stConfig.astMultiMasterAxisLatched[2].nIndex].stConfig.afMultiSlaveAxisRatio[GVL.iAxis] := _stAxis.Axis.PlcToNc.GearRatio2;
    _stAxis.stStatus.bCoupledGear2 := TRUE;
ELSE
    _stAxis.stStatus.bCoupledGear2 := FALSE;
END_IF

IF _stAxis.Axis.Status.Coupled AND _stAxis.Axis.PlcToNc.GearRatio3 <> 0 AND _stAxis.stConfig.astMultiMasterAxisLatched[3].nIndex <> 0 THEN
    GVL.astAxes[_stAxis.stConfig.astMultiMasterAxisLatched[3].nIndex].stConfig.afMultiSlaveAxisRatio[GVL.iAxis] := _stAxis.Axis.PlcToNc.GearRatio3;
    _stAxis.stStatus.bCoupledGear3 := TRUE;
ELSE
    _stAxis.stStatus.bCoupledGear3 := FALSE;
END_IF

IF _stAxis.Axis.Status.Coupled AND _stAxis.Axis.PlcToNc.GearRatio4 <> 0 AND _stAxis.stConfig.astMultiMasterAxisLatched[4].nIndex <> 0 THEN
    GVL.astAxes[_stAxis.stConfig.astMultiMasterAxisLatched[4].nIndex].stConfig.afMultiSlaveAxisRatio[GVL.iAxis] := _stAxis.Axis.PlcToNc.GearRatio4;
    _stAxis.stStatus.bCoupledGear4 := TRUE;
ELSE
    _stAxis.stStatus.bCoupledGear4 := FALSE;
END_IF
END_METHOD

METHOD mStatus_NewCommand : BOOL
VAR
    i: UINT;
END_VAR
fbExecuteRTrig(CLK := _stAxis.stControl.bExecute);
IF fbExecuteRTrig.Q THEN
    _stAxis.stStatus.bDone := FALSE;
    _stAxis.stStatus.bCommandAborted := FALSE;

    //On a new motion command, clear the errorID
    CASE _stAxis.stControl.eCommand OF
            E_MotionFunctions.eMoveAbsolute,
            E_MotionFunctions.eMoveRelative,
            E_MotionFunctions.eMoveVelocity,
            E_MotionFunctions.eMoveModulo,
            E_MotionFunctions.eGearInMultiMaster,
            E_MotionFunctions.eGearOut,
            E_MotionFunctions.eHome :
                _stAxis.stStatus.nErrorID := 0;
            E_MotionFunctions.eWriteParameter,
            E_MotionFunctions.eReadParameter,
            E_MotionFunctions.eReadCoEParameters,
            E_MotionFunctions.eWriteCoEParameters:
            // Nothing
    END_CASE
END_IF
END_METHOD

METHOD Run : BOOL
mStatus_AxisStatus();
mParameters_ReadNc();
mParameters_Init();
stMcStatusReadParameter := mParameters_ReadParameter();
stMcStatusWriteParameter := mParameters_WriteParameter();
stMcStatusReadWriteCoE := mParameters_ReadWriteCoE();

mControl_LimitHitTimer();
mControl_LimitLinking();
stMcStatusCommandHandler := mControl_CommandHandler(
    bAxisPermittedToMove := _stAxis.stStatus.bAxisReadyToMove
        AND (_stAxis.stStatus.bFwEnabled OR _stAxis.stStatus.bBwEnabled),
    bPermitRequired :=
        _stAxis.stConfig.bAutoEnable
        OR _stAxis.stConfig.stAirpadBrake.bAirpadConnected
        OR _stAxis.stConfig.stAirpadBrake.bExternalBrakeConnected,
    bWaitingForMovePermit => _stAxis.stStatus.bCommandHandlerBufferingCommand,
    bMovePermit => _stAxis.stStatus.bCommandHandlerMovePermit,
    bReleaseMoveCmd => _stAxis.stStatus.bCommandHandlerReleasedMoveCmd);

stMcStatusPower := mControl_Power();

stMcStatusAirpad := mControl_Airpad(
    bMoveRequest := (_stAxis.stStatus.bCommandHandlerBufferingCommand
            OR _stAxis.stStatus.bCommandHandlerMovePermit
            OR _stAxis.stStatus.bCommandHandlerReleasedMoveCmd
            OR _stAxis.stStatus.bMoving)
        AND _stAxis.stStatus.bEnabled,
    bManualControl := _stAxis.stConfig.bAirpadManualControl,
    bManualPressureOn := _stAxis.stControl.bAirpadManualPressureOn,
    bReady => _stAxis.stStatus.bAirpadReady);

stMcStatusHalt := mMove_Halt();
stMcStatusStop := mMove_Stop();
stMcStatusReset := mControl_Reset();

stMcStatusMoveAbsolute := mMove_MoveAbsolute();
stMcStatusMoveRelative := mMove_MoveRelative();
stMcStatusMoveModulo := mMove_MoveModulo();
stMcStatusMoveVelocity := mMove_MoveVelocity();

stMcStatusGearInMultiMaster := mControl_GearInMultiMaster();
stMcStatusGearOut := mControl_GearOut();

stMcStatusHome := mControl_Home();
stMcStatusBacklash := mControl_BacklashCompensation();

mStatus_NewCommand();
mStatus_Done();
mStatus_Error();
mStatus_InVelocity();
mStatus_CommandAborted();
_stAxis.stStatus.bBusy := mStatus_Busy();

EndOfCycle();
END_METHOD

PROPERTY stAxis : REFERENCE TO ST_AxisStruct
GET
stAxis REF= _stAxis;
END_GET
SET
_stAxis REF= stAxis;
END_SET
END_PROPERTY

END_FUNCTION_BLOCK

(* stored: Version 1.1.0.1
   POU FB_Axis: Id {beb60ab5-3bf2-0ae6-2037-f6d7e95a54b2}, SpecialFunc None
   Folder Control Methods: Id {c04e3e71-df24-0c4d-24b3-0aa19beb5b98}
   Folder Move Methods: Id {7637a174-c6eb-0da0-035a-7859ff006307}
   Folder Parameter Methods: Id {0fd27029-80d7-0d11-00e5-53d35724f1e8}
   Folder Status Methods: Id {8b59c6d7-3154-0e16-17b0-adcee2a0fc0f}
   Method EndOfCycle: Id {17524686-ff67-093e-3170-68964424d952}
   Method FB_init: Id {7ba0679f-ba8c-04d6-2152-f3231608cada}
   Method mControl_Airpad: Id {ec15769e-bbb8-0e4f-2638-9a7ccf63a25a}
   Method mControl_BacklashCompensation: Id {7107def5-ab6b-4951-863c-ccb3332d09d0}
   Method mControl_CommandHandler: Id {e4d415b3-33e2-0dab-1c34-04ed19023ade}
   Method mControl_ExternalBrake: Id {18ae79d4-85f5-0b8b-295a-ce90fc10f203}
   Method mControl_GearInMultiMaster: Id {7fc6d7a3-d42e-082e-332f-6abb17a6993e}
   Method mControl_GearOut: Id {1a5d2a0e-b81e-05b7-128d-5441f745907d}
   Method mControl_Home: Id {e7af0009-2f0b-0533-14d3-01b7d1874089}
   Method mControl_LimitHitTimer: Id {aac12074-ac2a-0993-05d9-b07faf70a873}
   Method mControl_LimitLinking: Id {28dddaf4-5369-0f3d-3c19-e3203d089e45}
   Method mControl_Power: Id {173f47fd-8a32-061e-2710-dce09d214d5b}
   Method mControl_Reset: Id {47f157c5-4fc8-0129-1c83-e659b71f8d37}
   Method mControl_TemperatureDisable: Id {a3234b7e-c99d-062f-2bbc-0982ac3ba282}
   Method mMove_Halt: Id {6e5dc22a-93e5-0120-008e-c508dd3989a9}
   Method mMove_MoveAbsolute: Id {6fddea8b-6d90-0fcc-2fdb-f5848d0817e2}
   Method mMove_MoveModulo: Id {f2bd8998-de45-0d9e-094c-0f21148a53b8}
   Method mMove_MoveRelative: Id {920dfedc-5c39-0e10-2be5-ecd6cce45da1}
   Method mMove_MoveVelocity: Id {2012a7b9-3d4f-08a7-33ac-a61d1acbd220}
   Method mMove_Stop: Id {580489a7-2144-0417-1656-bbc05af70ea7}
   Method mParameters_Init: Id {b94f4f04-02f5-00e2-1b47-81c18323a22e}
   Method mParameters_ReadNc: Id {6a2fb2fe-4cf7-03c3-0125-6e29359189a6}
   Method mParameters_ReadParameter: Id {60832699-55bc-043c-0cc0-4588cc7671e4}
   Method mParameters_ReadWriteCoE: Id {18f1550d-9340-4c35-816f-9023e1a97d47}
   Method mParameters_WriteParameter: Id {35a7c0ca-fdb5-465b-bd2a-42d607d9d72f}
   Method mStatus_AxisStatus: Id {6f0fec7d-27eb-00a8-18ec-af8d2df08244}
   Method mStatus_Busy: Id {41cf8366-0cbd-0f66-1e94-c9cc649849e7}
   Method mStatus_CommandAborted: Id {bcc908ba-00d1-061e-3ad8-e55a008deea3}
   Method mStatus_Done: Id {30b1d141-f7f0-0f00-2392-e4a3297bc4de}
   Method mStatus_Error: Id {072dc844-d4a9-0013-2e1e-f8d483107af4}
   Method mStatus_InVelocity: Id {300aae24-771f-08dd-22d3-a7e40414c3f7}
   Method mStatus_MultiGearing: Id {01b5ff71-e50a-0927-3f2f-4b0eddb7a326}
   Method mStatus_NewCommand: Id {95f7ac24-6eb9-0574-2499-da5c8ba45407}
   Method Run: Id {f4bb1bcc-b125-0a55-0aa6-fd00d78c99eb}
   Property stAxis: Id {6d5a6a07-8a3d-0159-072d-237a7e274fb7}
   Get Get: Id {4c6b0d2f-5bf4-0731-339f-cd189800c793}
   Set Set: Id {e0b65274-482d-0e17-2213-ff4e84fc47db} *)
